// TIA Portal V17 export
// export: Created 2024-06-14T09:52:42.7273844Z, ExportSetting WithDefaults, DisplayName Totally Integrated Automation Portal, DisplayVersion V17, DisplayName TIA Portal Openness, DisplayVersion V17, DisplayName TIA Portal Version Control Interface, DisplayVersion V17, DisplayName Simotion SCOUT TIA, DisplayVersion 5.4.3.0, DisplayName SINAMICS Startdrive Advanced, DisplayVersion V17 SP1 Update 1, DisplayName SINAMICS Startdrive G110M, G120, G120C, G120D, G120P, G115D, DisplayVersion V17 SP1 Update 1, DisplayName SINAMICS Startdrive G130, G150, S120, S150, SINAMICS MV, S210, DisplayVersion V17 SP1 Update 1, DisplayName STEP 7 Professional, DisplayVersion V17, DisplayName STEP 7 Safety, DisplayVersion V17, DisplayName WinCC Professional, DisplayVersion V17
DATA_BLOCK "MODBUS_DATA_WRITE"   // DB102
{ S7_Optimized_Access := 'FALSE' }
VERSION : 0.1
// stored: AutoNumber false, DBAccessibleFromOPCUA true, IsOnlyStoredInLoadMemory false, IsWriteProtectedInAS false
   VAR
      MOD_WR_DEV_STN4 : Array[1..6] of "MODBUS_WRITE";
      MOD_WR_DEV_STN5 : Array[1..6] of "MODBUS_WRITE";
      MOD_WR_DEV_CHECK_SCALE_1 { S7_SetPoint := 'True'} : "MODBUS_WRITE";
      MOD_WR_DEV_CORRECTION_SCALE { S7_SetPoint := 'True'} : "MODBUS_WRITE";
   END_VAR
BEGIN
END_DATA_BLOCK
